// TIA Portal V20 export
DATA_BLOCK "DB_LaserMeasureZoneSwitch"   // DB91
// stored: InstanceOfName FB_LaserMeasureZoneSwitch, InstanceOfType FB
"FB_LaserMeasureZoneSwitch"
   // VAR RETAIN
   //    sMeasure1 : Bool;
   //    sMeasure2 : Bool;
   //    sLaser1 : Bool;
   //    sLaser2 : Bool;
   //    sLaserArea1Req : Bool;
   //    sLaserArea2Req : Bool;
   //    sCuttingArea1Req : Bool;
   //    sCuttingArea2Req : Bool;
   //    sCutBusy : Bool;
   //    sCut1 : Bool;
   //    sCut2 : Bool;
   //    sX1Pos : Real;
   //    sX2Pos : Real;
   // END_VAR
   // VAR
   //    sRT_GateCut1 : R_TRIG;
   //    sRT_GateCut2 : R_TRIG;
   // END_VAR
   // VAR RETAIN
   //    sCondDegageAxe : Bool;
   //    sRefAxisActive : Bool;
   // END_VAR
BEGIN
END_DATA_BLOCK
